// TIA Portal V20 export
TYPE "LDrive_typeKistlerPressDataRecv"
// stored: IsFailsafeCompliant false
   STRUCT
      systemFixed : Struct
         Start : Bool;   // Mirrored Start Measuring
         TareY : Bool;   // Mirrored Channel Y Tare or Reset Piezo
         ZeroX : Bool;   // Mirrored Channel X zeros
         STestX : Bool;   // Mirrored Trigger sensor test for sensor X
         STestY : Bool;   // Mirrored Trigger sensor test for sensor Y
         ZeroExtendedX : Bool;
         MasterMeas : Bool;   // Mirrored Master measurement
         IncZero : Bool;   // Mirrored Zeros incremental sensor
         AckAdminGlobal : Bool;
         AckAdmin : Bool;   // Mirrored Acknowledgment with Admin rights (e.g., corresponding
         reserved1 : Bool;
         Access : Bool;   // Mirrored Allows the PLC to give the operator access rights
         Auto : Bool;   // Mirrored Auto, no editing of setup is possible
         StatReset : Bool;   // Mirrored statistics reset
         StatDisable : Bool;   // Deactivate mirrored statistics
         TaraExtendedY : Bool;
         MP : Byte;   // Mirrored measurement program choice
         reserved2 : Bool;
         reserved3 : Bool;
         resetSnGenerator : Bool;
         reserved4 : Bool;
         reserved5 : Bool;
         brakeTestActive : Bool;
         mirrorExportpvtStart : Bool;
         reserved6 : Bool;
         UNI_0 : Bool;   // Mirrored input signal UNI
         UNI_1 : Bool;   // Mirrored input signal UNI
         UNI_2 : Bool;   // Mirrored input signal UNI
         UNI_3 : Bool;   // Mirrored input signal UNI
         UNI_4 : Bool;   // Mirrored input signal UNI
         UNI_5 : Bool;   // Mirrored input signal UNI
         UNI_6 : Bool;   // Mirrored input signal UNI
         UNI_7 : Bool;   // Mirrored input signal UNI
         ReservedByte1 : Byte;
         Ready : Bool;   // Already
         OkTotal : Bool;   // Results GOOD
         NOkTotal : Bool;   // Results BAD
         NoPass : Bool;   // NO-PASS
         Reserved7 : Bool;
         Reserved8 : Bool;
         Warn : Bool;
         Alarm : Bool;
         S1 : Bool;   // Switching signal S1
         S2 : Bool;   // Switching signal S2
         Reserved9 : Bool;
         Reserved10 : Bool;
         Reserved11 : Bool;
         Reserved12 : Bool;
         Reserved13 : Bool;
         maxGradientStop : Bool;
         O_UNI_0 : Bool;
         O_UNI_1 : Bool;
         O_UNI_2 : Bool;
         O_UNI_3 : Bool;
         O_UNI_5 : Bool;
         O_UNI_4 : Bool;
         O_UNI_6 : Bool;
         O_UNI_7 : Bool;
         DriveEnable : Bool;   // Mirrored enable drive
         RunSequence : Bool;   // Mirrored command process of the sequence
         ReturnToHomePos : Bool;   // Mirrored command movement on base setting (MP-specific)
         DriveToRefPos : Bool;   // Mirrored command movement to reference position
         JogFW : Bool;   // Mirrored command jogging forwards
         JogBW : Bool;   // Mirrored command jogging backwards
         WaitRequest : Bool;   // Output is set through sequence object Wait. Sequencewaits for continuation through acknowledgment.
         BraketestDone : Bool;   // Brake test performed
         SequenceStopped : Bool;   // Sequence/command stopped
         SequenceEnd : Bool;   // Sequence/command ended
         OnlineEO_NOk : Bool;   // NOK for online evaluation of a corresponding EOs.Measurement ends
         StopViaExternalStop : Bool;   // External stop was set in sequence object
         SequenceError : Bool;   // Sequence/command error
         DriveEnabled : Bool;   // Enable drive set (current status of the enable)
         HomePosReached : Bool;   // Home position reached (NC joining module is in MP-specific)
         RefPosReached : Bool;   // Reference position reached (NC joining module is in
         Standstill : Bool;   // Standstill
         "Braketest Required" : Bool;   // Brake test required
         ServoWarn : Bool;   // Warning message on the servo amplifier pending
         ServoError : Bool;   // Alarm message on the servo amplifier pending
         SMES_Active : Bool;   // Safety status SMES active
         SMST2_Active : Bool;   // Safety status SMST2 active
         SMM1_Active : Bool;   // Safety status SMM1 active
         User_Mode_Active : Bool;   // Output is active (1) when the monitoring of the control
         Current_Sequence : Byte;   // Mirrored selection sequence Main, Sub1 ... 3
         Current_Label : Byte;   // Active label in thw sequence
         Cfg_MP : Byte;   // Mirrored measurement program choice of the input telegram
         jogToPosition : Bool;
         jogPosiitonReached : Bool;
         Reserved14 : Bool;
         Reserved15 : Bool;
         Reserved16 : Bool;
         Reserved17 : Bool;
         Reserved18 : Bool;
         Reserved19 : Bool;   // Mirrored bit of the input telegram
         CFG_ADR : Byte;   // Mirror CFG-ADR (up V 1.2.x.)
         CFG_Length : Byte;   // Mirror CFG-LENGTH (up V 1.2.x.)
         SelectedPage : Byte;   // Mirrored page select of the input telegram
         TransmissionFault : Bool;   // Error flag for transmission error.
         ACK : Bool;   // Acknowlage for strobe
         deviceavailable : Bool;
         Reserved20 : Bool;
         ChangedSelectedMP : Bool;   // Change flags of the measurement program changed.
         Reserved21 : Bool;
         ChangedSelectedGlobal : Bool;   // Change flags of global settings changed.
         backupComplete : Bool;
      END_STRUCT;
      userDefinedOutData : Array[20..219] of Byte;
   END_STRUCT;
END_TYPE
